Yaskawa INFORM job: WORKPIECE2.JBI

/JOB
//NAME WORKPIECE2
///FOLDERNAME INNE
//POS
///NPOS 10,10,0,0,0,0
///TOOL 0
///POSTYPE PULSE
///PULSE
C00000=34846,18001,86937,93778,55325,-59342
C00001=34431,-29522,5152,76593,58706,-45262
C00002=35202,-53816,-63523,62971,69519,-31037
C00003=114669,-93784,-99435,114651,-90398,-47027
C00004=113744,-63439,-13119,111243,-76195,-30802
C00005=109933,-121014,-87533,113021,-71100,-39893
C00006=115817,3588,31827,-1404,92004,-1585
C00007=147487,12091,39236,7520,90657,8603
C00008=193736,9628,36810,-20992,59161,-53276
C00009=118034,5626,33845,-770,91837,-869
BC00000=3493,452410,917391
BC00001=3492,452410,1075223
BC00002=3492,452410,1075223
BC00003=624,80186,893567
BC00004=624,192218,869947
BC00005=9,368120,826334
BC00006=298495,436540,859658
BC00007=298495,436540,859658
BC00008=298495,436540,859658
BC00009=297811,104835,859658
//INST
///DATE 2023/10/04 15:16
///ATTR SC,RW
///GROUP1 RB1,BS1
NOP
'LEFT_SIDE
MOVJ C00000 BC00000 VJ=0.78 PL=0  //POINT1
MOVJ C00001 BC00001 VJ=0.78 PL=0  //POINT2
MOVJ C00002 BC00002 VJ=0.78 PL=0  //POINT3
'BACK_SIDE
MOVJ C00003 BC00003 VJ=0.78 PL=0  //POINT1
MOVJ C00004 BC00004 VJ=0.78 PL=0  //POINT2
MOVJ C00005 BC00005 VJ=0.78 PL=0  //POINT3
'LEFT_2
MOVJ C00006 BC00006 VJ=0.78 PL=0  //POINT1
MOVJ C00007 BC00007 VJ=0.78 PL=0  //POINT2
MOVJ C00008 BC00008 VJ=0.78 PL=0  //POINT3
'RIGHT
MOVJ C00009 BC00009 VJ=0.78 PL=0  //POINT4
END
